FUNCTION F_SAFETY_StatusFB_TO_MUTING : ST_SAFETY_FBMUTING
VAR_INPUT
	stFBStatus						: ST_SAFETY_FBStatus; 	(* Struktura ogolna *)
END_VAR

F_SAFETY_StatusFB_TO_MUTING.uStatus.stStatusWords	:= stFBStatus;									(* Przepisanie *)
F_SAFETY_StatusFB_TO_MUTING.eState 					:= stFBStatus.BState;							(* Ustawienie enum *)
F_SAFETY_StatusFB_TO_MUTING.bGeneralError			:= stFBStatus.wDiagnosis <> 0;					(* General Error *)

END_FUNCTION

(* stored: Version 1.1.0.1, ProductVersion 3.1.4022.12
   POU F_SAFETY_StatusFB_TO_MUTING: Id {f4dc3dd4-688f-4575-ab03-8eae05e5fd86}, SpecialFunc None *)
